TYPE TestTableRow :
STRUCT
	timestamp : TIME;
	value1 : INT;
	value2 : REAL;
	description : STRING;
END_STRUCT
END_TYPE

(* stored: Version 1.1.0.1, ProductVersion 3.1.4024.12
   DUT TestTableRow: Id {ae7dc8aa-e613-0a47-31e9-ed08bd92dd4c} *)
